INTERFACE I_Disposable EXTENDS __SYSTEM.IQueryInterface

METHOD AddReference
VAR_INPUT
END_VAR
END_METHOD

METHOD Dispose
VAR_INPUT
END_VAR
END_METHOD

END_INTERFACE

(* stored: Version 1.1.0.1, ProductVersion 3.1.4024.11
   Itf I_Disposable: Id {6e581eb2-13c6-4ac8-9f8c-4e156ba44522}
   Method AddReference: Id {f5c19cb7-485e-4517-b570-a8c5dee2318e}
   Method Dispose: Id {9aa8024c-044f-4b2a-86d4-d160d511e242} *)
